PROGRAM POU_Control_Planta_1
VAR_INPUT
	X1: BOOL;
	X2:BOOL;
END_VAR

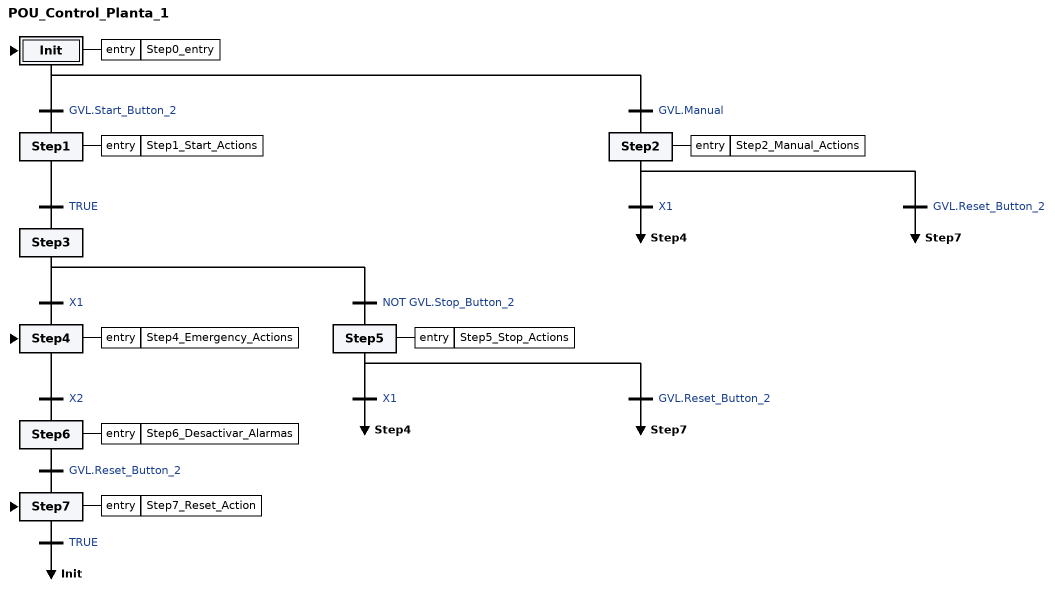
INITIAL_STEP Init:
    Step0_entry(P1);  // entry action
END_STEP
TRANSITION FROM Init TO Step1
    := GVL.Start_Button_2;
END_TRANSITION
STEP Step1:
    Step1_Start_Actions(P1);  // entry action
END_STEP
TRANSITION FROM Step1 TO Step3
    := TRUE;
END_TRANSITION
TRANSITION FROM Init TO Step2
    := GVL.Manual;
END_TRANSITION
STEP Step2:
    Step2_Manual_Actions(P1);  // entry action
END_STEP
TRANSITION FROM Step2 TO Step4
    := X1;
END_TRANSITION
TRANSITION FROM Step2 TO Step7
    := GVL.Reset_Button_2;
END_TRANSITION
STEP Step3:
END_STEP
TRANSITION FROM Step3 TO Step4
    := X1;
END_TRANSITION
STEP Step4:
    Step4_Emergency_Actions(P1);  // entry action
END_STEP
TRANSITION FROM Step4 TO Step6
    := X2;
END_TRANSITION
STEP Step6:
    Step6_Desactivar_Alarmas(P1);  // entry action
END_STEP
TRANSITION FROM Step6 TO Step7
    := GVL.Reset_Button_2;
END_TRANSITION
TRANSITION FROM Step3 TO Step5
    := NOT GVL.Stop_Button_2;
END_TRANSITION
STEP Step5:
    Step5_Stop_Actions(P1);  // entry action
END_STEP
TRANSITION FROM Step5 TO Step4
    := X1;
END_TRANSITION
TRANSITION FROM Step5 TO Step7
    := GVL.Reset_Button_2;
END_TRANSITION
STEP Step7:
    Step7_Reset_Action(P1);  // entry action
END_STEP
TRANSITION FROM Step7 TO Init
    := TRUE;
END_TRANSITION

ACTION Step0_entry:
GVL.Marcha := FALSE; // Se indica que la planta no puede funcionar
// Se indica mediante una luz que el siguiente botón a pulsar sería el de Start
GVL.Start_Button_2_Light := TRUE; 
GVL.Reset_Button_2_Light := FALSE;
// Se permite que la planta se mueva dentro del factory I/O
GVL.Factory_IO_Pause := FALSE;
GVL.Factory_IO_Reset := FALSE;
END_ACTION

ACTION Step1_Start_Actions:
GVL.Marcha := TRUE; // Se indica que la planta puede comenzar a funcionar
GVL.Emitter_1 := TRUE; // Se activa la emisión de piezas
GVL.Belt_Conveyor_2m_1 := 1; // Se activa la cinta de entrada
// Se indica mediante una luz que el siguiente botón a pulsar sería el de Stop
GVL.Start_Button_2_Light := FALSE; 
GVL.Stop_Button_2_Light := TRUE;
END_ACTION

ACTION Step2_Manual_Actions:
// Se indica mediante una luz que el siguiente botón a pulsar sería el de Reset
GVL.Start_Button_2_Light := FALSE;
GVL.Reset_Button_2_Light := TRUE;
END_ACTION

ACTION Step4_Emergency_Actions:
GVL.Marcha := FALSE; // Se indica que la planta no puede funcionar
// Se indica mediante una luz que el siguiente botón a pulsar sería el de Reset
GVL.Stop_Button_2_Light := FALSE;
GVL.Reset_Button_2_Light := TRUE;
//Se activan las alarmas
GVL.Alarm_Siren  := TRUE;
GVL.Warning_Light  := TRUE;
POU_Parada();
END_ACTION

ACTION Step5_Stop_Actions:
GVL.Emitter_1 := FALSE; // Se desactiva la emisión de piezas
GVL.Belt_Conveyor_2m_1 := 0; // Se desactiva la cinta de entrada
// Se indica mediante una luz que el siguiente botón a pulsar sería el de Reset
GVL.Stop_Button_2_Light := FALSE; 
GVL.Reset_Button_2_Light := TRUE;
END_ACTION

ACTION Step6_Desactivar_Alarmas:
//Se desactivan las alarmas
GVL.Alarm_Siren  := FALSE;
GVL.Warning_Light  := FALSE;
GVL.Factory_IO_Pause := FALSE;
END_ACTION

ACTION Step7_Reset_Action:
GVL.Factory_IO_Reset := TRUE;
//Se desactivan las alarmas
//GVL.Alarm_Siren  := FALSE;
//GVL.Warning_Light  := FALSE;
END_ACTION

END_PROGRAM

(* stored: Version 1.1.0.1, ProductVersion 3.1.4024.12
   POU POU_Control_Planta_1: Id {1ff5ca2a-77e7-44d4-8077-a3ce4d73de04}, SpecialFunc None
   Action Step0_entry: Id {7ce40ed1-dc4f-4787-a696-a8beae27949b}
   Action Step1_Start_Actions: Id {94b5dc4a-dc1f-45e3-ba69-a28bf4bf048e}
   Action Step2_Manual_Actions: Id {3520dc06-24ac-4646-b140-dce73f56815e}
   Action Step4_Emergency_Actions: Id {6fd7d359-e2a0-4309-8b5e-f809ee6743f9}
   Action Step5_Stop_Actions: Id {cf634960-712a-4288-acfd-7563677f0949}
   Action Step6_Desactivar_Alarmas: Id {20efe405-7d61-48a7-b473-d332e5391c43}
   Action Step7_Reset_Action: Id {0338bad7-279d-4171-b3a3-19c7706b75a3} *)
